(* IEC 61131-3 sources: CodesysTest/alpha/export/ObjectHandling/FB_CollectionHandlerActiveFaults.pou, 5 files *)

(* ---- FB_CollectionHandlerActiveFaults.pou.st ---- *)
(*#-#-#-#-#-#-#-#-#-#---Declaration---#-#-#-#-#-#-#-#-#-#-#-#-#*)

FUNCTION_BLOCK FB_CollectionHandlerActiveFaults
VAR_INPUT
END_VAR
VAR_OUTPUT
	totalObj : UINT;
	faultActive : BOOL;
	objNames : ARRAY[0..GlobalObjects.MAX_FAULTS] OF STRING;
	collection : ARRAY[0..GlobalObjects.MAX_FAULTS] OF IFault;
END_VAR
VAR

	_arrayOver : BOOL;
	_overObj : INT;
END_VAR(*#-#-#-#-#-#-#-#-#-#---Implementation---#-#-#-#-#-#-#-#-#-#-#-#-#*)

//	Function Block: FB_CollectionHandlerActiveFaults
//	Description: This collection handler adds and removes active faults to an array
//				 The add and remove methods are called from FB_Fault
//	Created by:
//	Created Date: Friday, September 7, 2018

(* ---- AckAll.m.st ---- *)
(*#-#-#-#-#-#-#-#-#-#---Declaration---#-#-#-#-#-#-#-#-#-#-#-#-#*)

METHOD AckAll
VAR_INPUT
END_VAR
VAR
	_cast : IFault;
	_fault : IFault;
	_j : UINT;
END_VAR(*#-#-#-#-#-#-#-#-#-#---Implementation---#-#-#-#-#-#-#-#-#-#-#-#-#*)

// For each active fault in the array, ack it.
FOR _j:= 0 TO totalObj - 1 DO
	IF (__QUERYINTERFACE(Collection[_j], _cast)) THEN
		_cast.Ack();
	ELSE
		RETURN;
	END_IF
END_FOR

(* ---- AddObject.m.st ---- *)
(*#-#-#-#-#-#-#-#-#-#---Declaration---#-#-#-#-#-#-#-#-#-#-#-#-#*)

METHOD AddObject
VAR_INPUT
	obj   : IFault;
END_VAR
VAR
	_j : UINT;
END_VAR(*#-#-#-#-#-#-#-#-#-#---Implementation---#-#-#-#-#-#-#-#-#-#-#-#-#*)

// Add the active fault to the array
FOR _j:= 0 TO totalObj DO
	IF Collection[_j] = obj THEN
		// object pointer matches - it's already in here
		RETURN;
	END_IF
END_FOR

//
IF totalObj < GlobalObjects.MAX_FAULTS THEN
	Collection[totalObj]:= obj;
	objNames[totalObj]:= obj.InstanceName;
	totalObj:= totalObj + 1;
ELSE
	_ArrayOver:= TRUE;
	_OverObj:= _OverObj + 1;
END_IF
faultActive := TRUE;

(* ---- ContainsObject.m.st ---- *)
(*#-#-#-#-#-#-#-#-#-#---Declaration---#-#-#-#-#-#-#-#-#-#-#-#-#*)

METHOD ContainsObject : BOOL
VAR_INPUT
	objName : STRING;
END_VAR
VAR
	_i : UINT;
END_VAR
(*#-#-#-#-#-#-#-#-#-#---Implementation---#-#-#-#-#-#-#-#-#-#-#-#-#*)

// Add the active fault to the array
FOR _i := 0 TO totalObj DO
	IF objNames[_i] = objName THEN
		ContainsObject := TRUE;
		RETURN;
	END_IF
END_FOR
ContainsObject := FALSE;

(* ---- RemoveObject.m.st ---- *)
(*#-#-#-#-#-#-#-#-#-#---Declaration---#-#-#-#-#-#-#-#-#-#-#-#-#*)

METHOD RemoveObject
VAR_INPUT
	obj   : IFault;
END_VAR
VAR
	_i : UINT;
	_j : UINT;
END_VAR
(*#-#-#-#-#-#-#-#-#-#---Implementation---#-#-#-#-#-#-#-#-#-#-#-#-#*)

FOR _i:= 0 TO totalObj DO
	IF Collection[_i] = obj THEN
		// object pointer matches - get rid of it
		FOR _j := _i TO totalObj DO
			Collection[_j] := Collection[_j+1];
			objNames[_j]:= objNames[_j+1];
		END_FOR
		totalObj := totalObj - 1;
		IF totalObj = 0 THEN
			faultActive := FALSE;
		END_IF
		RETURN;
	END_IF
END_FOR
